{attribute 'linkalways'} 
{attribute 'no_explicit_call' := 'This FB is a CLASS and must be accessed using methods or properties'}
{attribute 'enable_dynamic_creation'}
FUNCTION_BLOCK _TcVnVector4_USINT EXTENDS AliasDatatypeBase
VAR
	localData : TcVnVector4_USINT;
	activeData : REFERENCE TO TcVnVector4_USINT REF= localData;
	aliasBaseDatatype : _Array0to3OfUSINT;
END_VAR

PROPERTY PUBLIC Address : PVOID
GET
Address := ADR(activeData);
END_GET
END_PROPERTY

METHOD PUBLIC ClearReference
VAR_INPUT
END_VAR
activeData REF= localData;
SetBaseDatatypeReference();
END_METHOD

METHOD PUBLIC Clone : I_Datatype
VAR
    pClone : POINTER TO _TcVnVector4_USINT;
END_VAR
pClone := __NEW(_TcVnVector4_USINT);
Clone := pClone^;
END_METHOD

METHOD FB_init : BOOL
VAR_INPUT
	bInitRetains : BOOL; // if TRUE, the retain variables are initialized (warm start / cold start)
	bInCopyCode : BOOL;  // if TRUE, the instance afterwards gets moved into the copy code (online change)
	//InitialValue : <type>; // if possible, not all values can be initialized
END_VAR
//localData := InitialValue; // if possible, not all values can be initialized
SetBaseDatatypeReference();
AddBaseDatatype(aliasBaseDatatype);
END_METHOD

PROPERTY PUBLIC Identifier : T_MAXSTRING
GET
Identifier := 'TcVnVector4_USINT';
END_GET
END_PROPERTY

METHOD PUBLIC MakeReferenceTo
VAR_INPUT
	ReferenceTarget : REFERENCE TO TcVnVector4_USINT;
END_VAR
activeData REF= ReferenceTarget;
SetBaseDatatypeReference();
END_METHOD

METHOD PROTECTED SetBaseDatatypeReference
VAR_INPUT
END_VAR
aliasBaseDatatype.MakeReferenceTo(activeData);
END_METHOD

PROPERTY PUBLIC Size : UDINT
GET
Size := SIZEOF(activeData);
END_GET
END_PROPERTY

METHOD TryMakeReferenceTo : BOOL
VAR_INPUT
	Target : I_Datatype;
END_VAR
VAR
	targetAsAlias : I_AliasDatatype;
	pTargetData : POINTER TO TcVnVector4_USINT;
END_VAR
IF NOT Target.TryResolveAsAliasDatatype(targetAsAlias) THEN
	RETURN;
END_IF

IF targetAsAlias.Identifier <> Identifier THEN
	RETURN;
END_IF

pTargetData := Target.Address;
activeData REF= pTargetData^;
SetBaseDatatypeReference();
TryMakeReferenceTo := TRUE;
END_METHOD

PROPERTY PUBLIC Value : REFERENCE TO TcVnVector4_USINT
GET
Value REF= activeData;
END_GET
END_PROPERTY

END_FUNCTION_BLOCK

(* stored: Version 1.1.0.1, ProductVersion 3.1.4024.13
   POU _TcVnVector4_USINT: Id {d88fd0b5-6846-061d-181d-9eb218cdbbf0}, SpecialFunc None
   Folder Core: Id {a21c1c4f-b8ff-04dc-193d-c2c084012e48}
   Folder Protected: Id {55481c2e-dded-01dc-3bfe-cb787456227f}
   Folder Customize: Id {9b70458d-a76f-0cb7-19f3-98a17a0ef990}
   Folder Constructor: Id {0fd1ba50-4bf7-0fb9-2d41-cbee32fcd01b}
   Property Address: Id {d88ae4d8-ae49-054b-2cfa-7182125789f0}
   Get Get: Id {693b883f-4d5c-0d92-0a94-147c2ff76d2a}
   Method ClearReference: Id {e2507e8d-5082-0c79-1113-e7b89ca0601c}
   Method Clone: Id {bedf673b-65af-050d-368a-a09946a15f0f}
   Method FB_init: Id {0503d5d4-8265-0cbf-3e96-c533729bdf08}
   Property Identifier: Id {cb0aee59-7184-0cfe-3152-06ab7a0a833a}
   Get Get: Id {94abfa1f-870e-0175-22b3-e66ce3bc85ec}
   Method MakeReferenceTo: Id {f35fe290-55c4-0c88-3a0b-599b4099300d}
   Method SetBaseDatatypeReference: Id {0a5cbf4e-6a9a-06ee-35ec-21539c0e7c58}
   Property Size: Id {a541e729-1c5a-09a1-0aa3-b5474360a015}
   Get Get: Id {5e426851-f2f3-01a9-207f-1afb199ec1da}
   Method TryMakeReferenceTo: Id {6b24764b-de88-0ea5-04f9-4ba4642b0e5f}
   Property Value: Id {c3a29cf3-2dee-0687-0ef9-2aec8675dbf3}
   Get Get: Id {e7c9faf6-7347-09ba-234b-c284eccf2549} *)
